TYPE ST_Test1 EXTENDS ST_Base :
STRUCT
	nTest4 : INT;
	stBase : ST_Base;
END_STRUCT
END_TYPE

(* stored: Version 1.1.0.1
   DUT ST_Test1: Id {6e0179cd-d933-42eb-86ef-958c2772dfc6} *)
